% RSLogix 500 project I2A-JOB-15-MITCH_BAK108.RSS, saved by version 10.00.00.00 %
PROJECT "ML01B"    % processor: Bul.1763 MicroLogix 1100 Series B %

PROGRAM FILES
  LAD 2   15 rungs

DATA FILES
  O0 OUTPUT  4 elements
  I1 INPUT  6 elements
  S2 STATUS  66 elements
  B3 BINARY  1 elements
  T4 TIMER  1 elements
  C5 COUNTER  1 elements
  R6 CONTROL  1 elements
  N7 INTEGER  1 elements
  F8 FLOAT  1 elements

LADDER 2
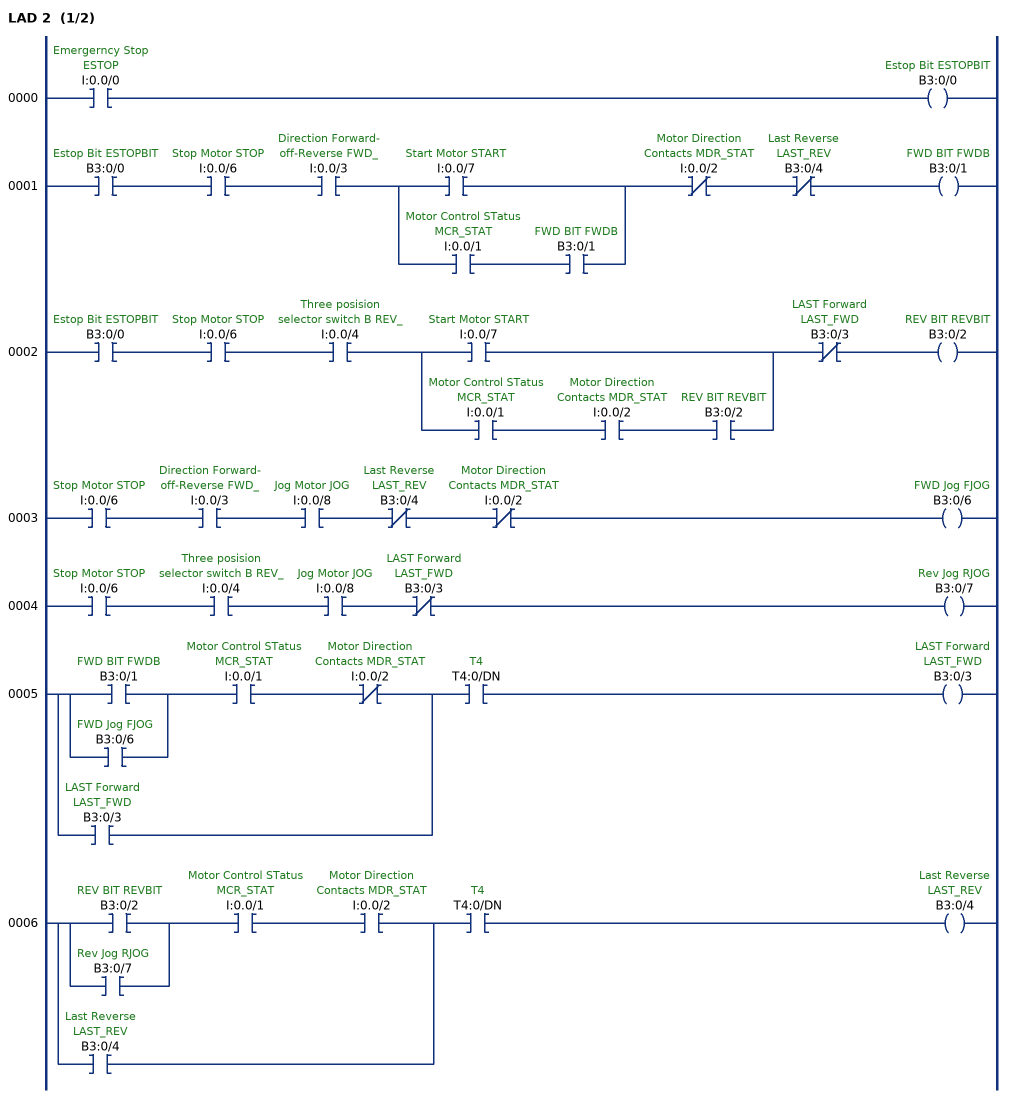
% Rung: 0 %
SOR XIC I:0.0/0 OTE B3:0/0 EOR
%   I:0.0/0  ESTOP  "Emergerncy Stop" %
%   B3:0/0  ESTOPBIT  "Estop Bit" %
% Rung: 1 %
SOR XIC B3:0/0 XIC I:0.0/6 XIC I:0.0/3 BST XIC I:0.0/7 NXB XIC I:0.0/1 XIC B3:0/1 BND XIO I:0.0/2 XIO B3:0/4 OTE B3:0/1 EOR
%   B3:0/0  ESTOPBIT  "Estop Bit" %
%   I:0.0/6  STOP  "Stop Motor" %
%   I:0.0/3  FWD_  "Direction Forward- off-Reverse" %
%   I:0.0/7  START  "Start Motor" %
%   I:0.0/1  MCR_STAT  "Motor Control STatus" %
%   B3:0/1  FWDB  "FWD BIT" %
%   I:0.0/2  MDR_STAT  "Motor Direction Contacts" %
%   B3:0/4  LAST_REV  "Last Reverse" %
% Rung: 2 %
SOR XIC B3:0/0 XIC I:0.0/6 XIC I:0.0/4 BST XIC I:0.0/7 NXB XIC I:0.0/1 XIC I:0.0/2 XIC B3:0/2 BND XIO B3:0/3 OTE B3:0/2 EOR
%   B3:0/0  ESTOPBIT  "Estop Bit" %
%   I:0.0/6  STOP  "Stop Motor" %
%   I:0.0/4  REV_  "Three posision selector switch B" %
%   I:0.0/7  START  "Start Motor" %
%   I:0.0/1  MCR_STAT  "Motor Control STatus" %
%   I:0.0/2  MDR_STAT  "Motor Direction Contacts" %
%   B3:0/2  REVBIT  "REV BIT" %
%   B3:0/3  LAST_FWD  "LAST Forward" %
% Rung: 3 %
SOR XIC I:0.0/6 XIC I:0.0/3 XIC I:0.0/8 XIO B3:0/4 XIO I:0.0/2 OTE B3:0/6 EOR
%   I:0.0/6  STOP  "Stop Motor" %
%   I:0.0/3  FWD_  "Direction Forward- off-Reverse" %
%   I:0.0/8  JOG  "Jog Motor" %
%   B3:0/4  LAST_REV  "Last Reverse" %
%   I:0.0/2  MDR_STAT  "Motor Direction Contacts" %
%   B3:0/6  FJOG  "FWD Jog" %
% Rung: 4 %
SOR XIC I:0.0/6 XIC I:0.0/4 XIC I:0.0/8 XIO B3:0/3 OTE B3:0/7 EOR
%   I:0.0/6  STOP  "Stop Motor" %
%   I:0.0/4  REV_  "Three posision selector switch B" %
%   I:0.0/8  JOG  "Jog Motor" %
%   B3:0/3  LAST_FWD  "LAST Forward" %
%   B3:0/7  RJOG  "Rev Jog" %
% Rung: 5 %
SOR BST BST XIC B3:0/1 NXB XIC B3:0/6 BND XIC I:0.0/1 XIO I:0.0/2 NXB XIC B3:0/3 BND XIC T4:0/DN OTE B3:0/3 EOR
%   B3:0/1  FWDB  "FWD BIT" %
%   B3:0/6  FJOG  "FWD Jog" %
%   I:0.0/1  MCR_STAT  "Motor Control STatus" %
%   I:0.0/2  MDR_STAT  "Motor Direction Contacts" %
%   B3:0/3  LAST_FWD  "LAST Forward" %
%   T4:0/DN  T4 %
% Rung: 6 %
SOR BST BST XIC B3:0/2 NXB XIC B3:0/7 BND XIC I:0.0/1 XIC I:0.0/2 NXB XIC B3:0/4 BND XIC T4:0/DN OTE B3:0/4 EOR
%   B3:0/2  REVBIT  "REV BIT" %
%   B3:0/7  RJOG  "Rev Jog" %
%   I:0.0/1  MCR_STAT  "Motor Control STatus" %
%   I:0.0/2  MDR_STAT  "Motor Direction Contacts" %
%   B3:0/4  LAST_REV  "Last Reverse" %
%   T4:0/DN  T4 %

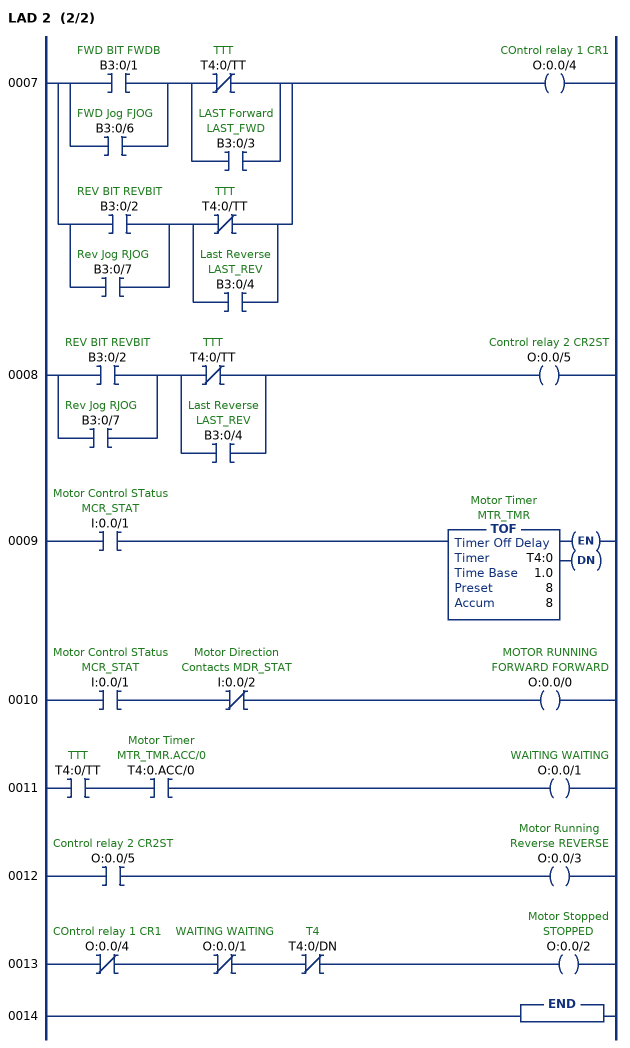
% Rung: 7 %
SOR BST BST XIC B3:0/1 NXB XIC B3:0/6 BND BST XIO T4:0/TT NXB XIC B3:0/3 BND NXB BST XIC B3:0/2 NXB XIC B3:0/7 BND BST XIO T4:0/TT NXB XIC B3:0/4 BND BND OTE O:0.0/4 EOR
%   B3:0/1  FWDB  "FWD BIT" %
%   B3:0/6  FJOG  "FWD Jog" %
%   T4:0/TT  TTT %
%   B3:0/3  LAST_FWD  "LAST Forward" %
%   B3:0/2  REVBIT  "REV BIT" %
%   B3:0/7  RJOG  "Rev Jog" %
%   B3:0/4  LAST_REV  "Last Reverse" %
%   O:0.0/4  CR1  "COntrol relay 1" %
% Rung: 8 %
SOR BST XIC B3:0/2 NXB XIC B3:0/7 BND BST XIO T4:0/TT NXB XIC B3:0/4 BND OTE O:0.0/5 EOR
%   B3:0/2  REVBIT  "REV BIT" %
%   B3:0/7  RJOG  "Rev Jog" %
%   T4:0/TT  TTT %
%   B3:0/4  LAST_REV  "Last Reverse" %
%   O:0.0/5  CR2ST  "Control relay 2" %
% Rung: 9 %
SOR XIC I:0.0/1 TOF T4:0 1.0 8 8 EOR
%   I:0.0/1  MCR_STAT  "Motor Control STatus" %
%   T4:0  MTR_TMR  "Motor Timer" %
% Rung: 10 %
SOR XIC I:0.0/1 XIO I:0.0/2 OTE O:0.0/0 EOR
%   I:0.0/1  MCR_STAT  "Motor Control STatus" %
%   I:0.0/2  MDR_STAT  "Motor Direction Contacts" %
%   O:0.0/0  FORWARD  "MOTOR RUNNING FORWARD" %
% Rung: 11 %
SOR XIC T4:0/TT XIC T4:0.ACC/0 OTE O:0.0/1 EOR
%   T4:0/TT  TTT %
%   T4:0  MTR_TMR  "Motor Timer" %
%   O:0.0/1  WAITING  "WAITING" %
% Rung: 12 %
SOR XIC O:0.0/5 OTE O:0.0/3 EOR
%   O:0.0/5  CR2ST  "Control relay 2" %
%   O:0.0/3  REVERSE  "Motor Running Reverse" %
% Rung: 13 %
SOR XIO O:0.0/4 XIO O:0.0/1 XIO T4:0/DN OTE O:0.0/2 EOR
%   O:0.0/4  CR1  "COntrol relay 1" %
%   O:0.0/1  WAITING  "WAITING" %
%   T4:0/DN  T4 %
%   O:0.0/2  STOPPED  "Motor Stopped" %
% Rung: 14 %
SOR END EOR

OTHER DOCUMENTED ADDRESSES
  B3:0/5  RUN  "RUn Bit"
  I:0.0/5  2PSSA  "2 position selector switch A"
  T4:1/TT  TT

DATA TABLE (non-zero values as saved)
DATA B3
% B3:0 % 0X0001
DATA T4
% .PRE .ACC %
% T4:0 % 8 8
DATA C5
% .PRE .ACC %
% C5:0 % 16 0
